PROGRAM LOGGER
VAR
	fbLogger	:	FB_Logger;
END_VAR

fbLogger();

END_PROGRAM

(* stored: Version 1.1.0.1, ProductVersion 3.1.4018.5
   POU LOGGER: Id {7711980f-2638-427e-8c10-3ab42f4b7695}, SpecialFunc None *)
